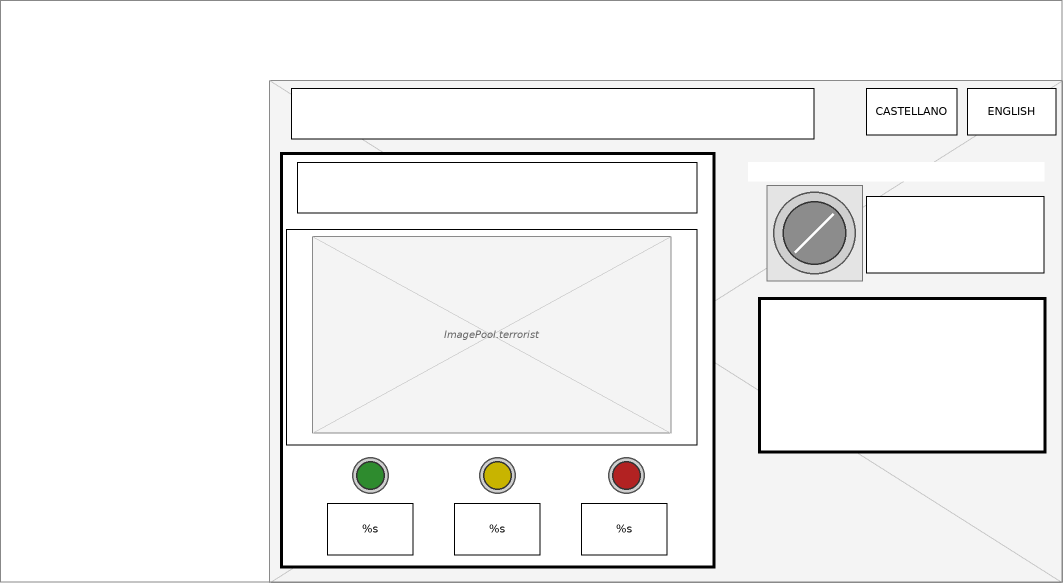
VISUALIZATION Visualization  // 1063x583
    Image (269,80 794x503), image: ImagePool.himcap
    RoundedRectangle (280,152 435x416)
    Rectangle (286,229 411x216)
    Image (312,236 359x197), image: ImagePool.terrorist
        p84334746: MAIN.HMI_CTRL.sImagenActual
    RotarySwitch (765,185 99x96), variable: MAIN.EMERGENCY_HDL.stSystem.inputs.iSwitch_HMI, behaviour: TOGGLE, style: Switch-RotarySwitch-Gray
    Rectangle (748,162 296x19), "%s", text list: 'TextList', text index: 5
    Lamp1 (349,453 43x45), variable: MAIN.stSystem.outputs.oLightGreen, style: Lamp-Lamp1-Green
    Lamp1 (476,453 43x45), variable: MAIN.stSystem.outputs.oLightOrange, style: Lamp-Lamp1-Yellow
    Lamp1 (605,453 43x45), variable: MAIN.stSystem.outputs.oLightRed, style: Lamp-Lamp1-Red
    RoundedRectangle (327,503 86x52), "%s", text list: 'TextList', text index: 2
    RoundedRectangle (454,503 86x52), "%s", text list: 'TextList', text index: 3
    RoundedRectangle (581,503 86x52), "%s", text list: 'TextList', text index: 4
    Rectangle (891,297 155x156)
    Rectangle (297,162 400x51), "%s", text list: 'TextList', text index: 1
    RoundedRectangle (967,88 89x47), "ENGLISH"
        OnMouseClick: ChangeLanguage ChangeLanguage=English
    RoundedRectangle (866,88 91x47), "CASTELLANO"
        OnMouseClick: ChangeLanguage ChangeLanguage=Spanish
    Rectangle (866,196 178x77), "%s", text list: 'TextList', text index: 0
    Rectangle (291,88 523x51), "%s", text list: 'TextList', text index: 9
    RoundedRectangle (758,297 288x156)
        toggle MAIN.EMERGENCY_HDL.stSystem.inputs.iAlarmButton_HMI
    Rectangle (753,360 291x34), "%s", text list: 'TextList', text index: 6
END_VISUALIZATION

(* stored: Version 1.1.0.1, ProductVersion 3.1.4026.12
   Visu Visualization: Id {f68d792a-53b6-48f5-87e2-be1b702acad6} *)
